(* IEC 61131-3 sources: Lasal/CPU_5344_V01/Class/multipleTrigger, 1 file *)

(* ---- multipleTrigger.st ---- *)
(*!
<Class
	Name               = "multipleTrigger"
	Revision           = "0.0"
	RealtimeTask       = "false"
	CyclicTask         = "true"
	DefCyclictime      = "10 ms"
	BackgroundTask     = "false"
	Sigmatek           = "false"
	OSInterface        = "false"
	HighPriority       = "false"
	Automatic          = "false"
	UpdateMode         = "Prescan"
	SharedCommandTable = "true"
	Objectsize         = "(284,120)">
	<Channels>
		<Server Name="typeAction" Visualized="false" Initialize="true" DefValue="1" WriteProtected="false" Retentive="false" Comment="1 means only positive triggers&#13;&#10;2 means only negative triggers&#13;&#10;else both triggers&#13;&#10;"/>
		<Client Name="client1" Required="true" Internal="false"/>
		<Client Name="client2" Required="false" Internal="false"/>
		<Client Name="client3" Required="false" Internal="false"/>
		<Client Name="client4" Required="false" Internal="false"/>
		<Client Name="input" Required="true" Internal="false"/>
	</Channels>
</Class>
*)
multipleTrigger : CLASS
  //Servers:
	typeAction 	: SvrChCmd_DINT;
  //Clients:
	input 	: CltCh_DINT;
	client1 	: CltCh_DINT;
	client2 	: CltCh_DINT;
	client3 	: CltCh_DINT;
	client4 	: CltCh_DINT;
  //Variables:
		oldInput 	: DINT;
  //Functions:

	FUNCTION VIRTUAL GLOBAL CyWork
		VAR_INPUT
			EAX 	: UDINT;
		END_VAR
		VAR_OUTPUT
			state (EAX) 	: UDINT := READY;
		END_VAR;
  //Tables:
	FUNCTION @STD
		VAR_OUTPUT
			ret_code	: CONFSTATES;
		END_VAR;
	FUNCTION GLOBAL TAB @CT_;
END_CLASS;

// JdK 22-7-2019: multipleTrigger created for Traffiroad/4284

// goal is to write changement of server to 4 clients

FUNCTION VIRTUAL GLOBAL multipleTrigger::CyWork
	VAR_INPUT
		EAX 	: UDINT;
	END_VAR
	VAR_OUTPUT
		state (EAX) 	: UDINT;(* := READY *)
	END_VAR

  input:=input.Read();

  IF input <> oldInput & (input=1 | typeAction<> 1) & (input=0 | typeAction<>2) THEN //only on positive/negative trigger
    client1:=client2:=client3:=client4:=input;
    client1.Write (client1);
    client2.Write (client2);
    client3.Write (client3);
    client4.Write (client4);
  END_IF;
  oldInput:= input;

END_FUNCTION
